// TIA Portal V20 export
DATA_BLOCK "Tippler_HMI"   // DB401
{ S7_Optimized_Access := 'TRUE' }
// stored: AutoNumber false, MemoryReserve 100
   VAR
      MT_Control : Bool;
      HMI_Control : Bool;
      Up : Bool;
      Down : Bool;
      MT_Arm_Selection : Int;
      Button_Up : Bool;
      Button_Down : Bool;
      Set_Angle : Int;
      MT_Button_Open : Bool;
      MT_Button_Close : Bool;
      MT_Button_Up : Bool;
      MT_Button_Down : Bool;
      Kip1_UP_maint : Bool;
      Kip1_Down_maint : Bool;
      Kip2_UP_maint : Bool;
      Kip2_Down_maint : Bool;
      Kip_Both_Up : Bool;
      Kip_Both_Down : Bool;
   END_VAR
BEGIN
END_DATA_BLOCK
